// TIA Portal V18 export
VAR_GLOBAL   // PLC tag table "25_ESP-EG3"
   "iESP-EG3" AT %I13.2 : Bool;
   "oESP-EG3" AT %Q12.5 : Bool;
END_VAR
